INTERFACE I_Alarm

PROPERTY AlarmId : DINT
GET
END_GET
END_PROPERTY

PROPERTY ArgStackMemoryPointer : POINTER TO BYTE
GET
END_GET
END_PROPERTY

PROPERTY ArgStackMemorySize : DINT
GET
END_GET
END_PROPERTY

END_INTERFACE

(* stored: Version 1.1.0.1, ProductVersion 3.1.4024.15
   Itf I_Alarm: Id {de3a4b9d-4f16-4f54-a6f5-7e2689dd293f}
   Property AlarmId: Id {c5a5d68f-cd0c-414a-9996-a847e04ecc98}
   Get Get: Id {de953d70-013d-44a7-82e0-2435ad613e94}
   Property ArgStackMemoryPointer: Id {4852cf3b-552a-4a1f-9267-4f27b52cc012}
   Get Get: Id {2a1d79db-762c-4aa7-8cbe-3e9bd2f7090c}
   Property ArgStackMemorySize: Id {19302f09-37fe-4fe1-ac4e-bd14a66e3108}
   Get Get: Id {bfc9c7aa-4e4e-4b09-a1ff-dab0ad1d6954} *)
